(* CODESYS project EX3.project

Project tree, tasks and I/O mapping:
  Device : CODESYS Control Win V3, 3S - Smart Software Solutions GmbH, order no. 305021, version 3.5.11.30
    application Application
      libraries: Standard, * (System)
      task MainTask (cyclic, interval t#20ms, priority 1) calls PLC_PRG
      task VISU_TASK (cyclic, interval 100 ms, priority 31) calls VisuElems.Visu_Prg
      program PLC_PRG [LD]
      visualisation Visualization
  text list GlobalTextList
*)

// Device/Application/PLC_PRG
PROGRAM PLC_PRG
VAR
	B1 : BOOL;          // BOMBA 
	L1 : BOOL;          // LAMPADA DE SINALIZACAO
	PT1 : BOOL;         // SENSOR DE PRESSAO
	BT1 : BOOL;         // BOTAO NA RETENTIVO
END_VAR
VAR // added by the converter: edge detectors and wires of the graphical bodies
    _w1 : BOOL;
END_VAR

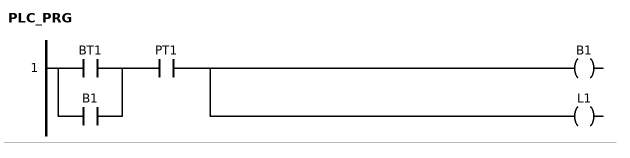
// NETWORK 1
_w1 := (BT1 OR B1) AND PT1;
B1 := _w1;
L1 := _w1;

END_PROGRAM

// Device/Application/Visualization
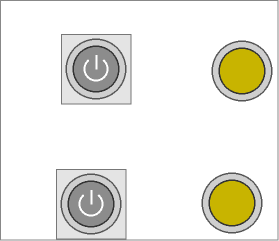
VISUALIZATION Visualization  // 279x241
    Lamp1 (207,36 70x70), variable: PLC_PRG.L1, style: Lamp-Lamp1-Yellow
    PowerSwitch (61,34 70x70), variable: PLC_PRG.BT1, behaviour: TAP, style: Switch-PowerSwitch-Gray
    Lamp1 (197,168 70x70), variable: PLC_PRG.B1, style: Lamp-Lamp1-Yellow
    PowerSwitch (56,169 70x70), variable: PLC_PRG.PT1, behaviour: TOGGLE, style: Switch-PowerSwitch-Gray
END_VISUALIZATION
